FUNCTION_BLOCK CU050ManualTask EXTENDS TcoTaskedService IMPLEMENTS ICUTask
VAR
END_VAR

Run();

(*~
	<docu>
		<summary>
			Main method of the sequener. Custom code needs to be placed here. The sequencer is executed by call of **Instance.Run()** method.
			This method is abstract, and it must be overridden in derived block.
		</summary>
	</docu>
~*)
METHOD PROTECTED Main : BOOL
Messenger.Notify('Running manual mode');
Station.Components.Group1.horizontalCylinder.Service();
END_METHOD

METHOD PROTECTED OnStart
Station.AutomatTask.Restore();
Station.GroundTask.Restore();
Station.GroundTask.CancelGround();
END_METHOD

PROPERTY Station : REFERENCE TO CU050
GET
VAR
    _station : POINTER TO CU050;
END_VAR
IF __QUERYPOINTER(Parent, _station) THEN // Check if _Parent is Station001
    Station REF= _station^;              // If the check is successful dereference a pointer. simlar to THIS^ or SUPER^
END_IF
END_GET
END_PROPERTY

END_FUNCTION_BLOCK

(* stored: Version 1.1.0.1
   POU CU050ManualTask: Id {f613db05-9014-442d-b92a-681bdad49089}, SpecialFunc None
   Method Main: Id {4c3dd489-b605-4a19-82dd-becc292d88df}
   Method OnStart: Id {aeadeb5a-295e-4b0e-bf8f-2dde1f3b6e99}
   Property Station: Id {fffabdf1-3e1c-4c1e-a9f0-120e10625bd9}
   Get Get: Id {49a059f4-9691-4dd7-b391-fbbc1cb3f267} *)
